// TIA Portal V17 export
// export: Created 2025-06-26T07:49:41.1534904Z, ExportSetting WithDefaults, DisplayName Totally Integrated Automation Portal, DisplayVersion V17 Update 8, DisplayName TIA Portal Openness, DisplayVersion V17 Update 8, DisplayName TIA Portal Version Control Interface, DisplayVersion V17, DisplayName STEP 7 Professional, DisplayVersion V17 Update 8, DisplayName STEP 7 Safety, DisplayVersion V17 Update 6, DisplayName WinCC Advanced, DisplayVersion V17 Update 8
FUNCTION "State2_Standby" : Void   // FC9, FBD
{ S7_Optimized_Access := 'TRUE' }
VERSION : 0.1
// stored: AutoNumber true, IsIECCheckEnabled false, SetENOAutomatically false, UDAEnableTagReadback false
   VAR_INPUT
      Active : Bool;
   END_VAR
   VAR_OUTPUT
      NextState : Bool;
      Stop : Bool;
   END_VAR
   VAR_TEMP
      NextStateConditions : Bool;
      PauseHere : Bool;
   END_VAR
   VAR_TEMP   // added for the SCL form of the ladder/FBD networks
      _w1 : Bool;
   END_VAR
BEGIN

REGION Network 1: State number
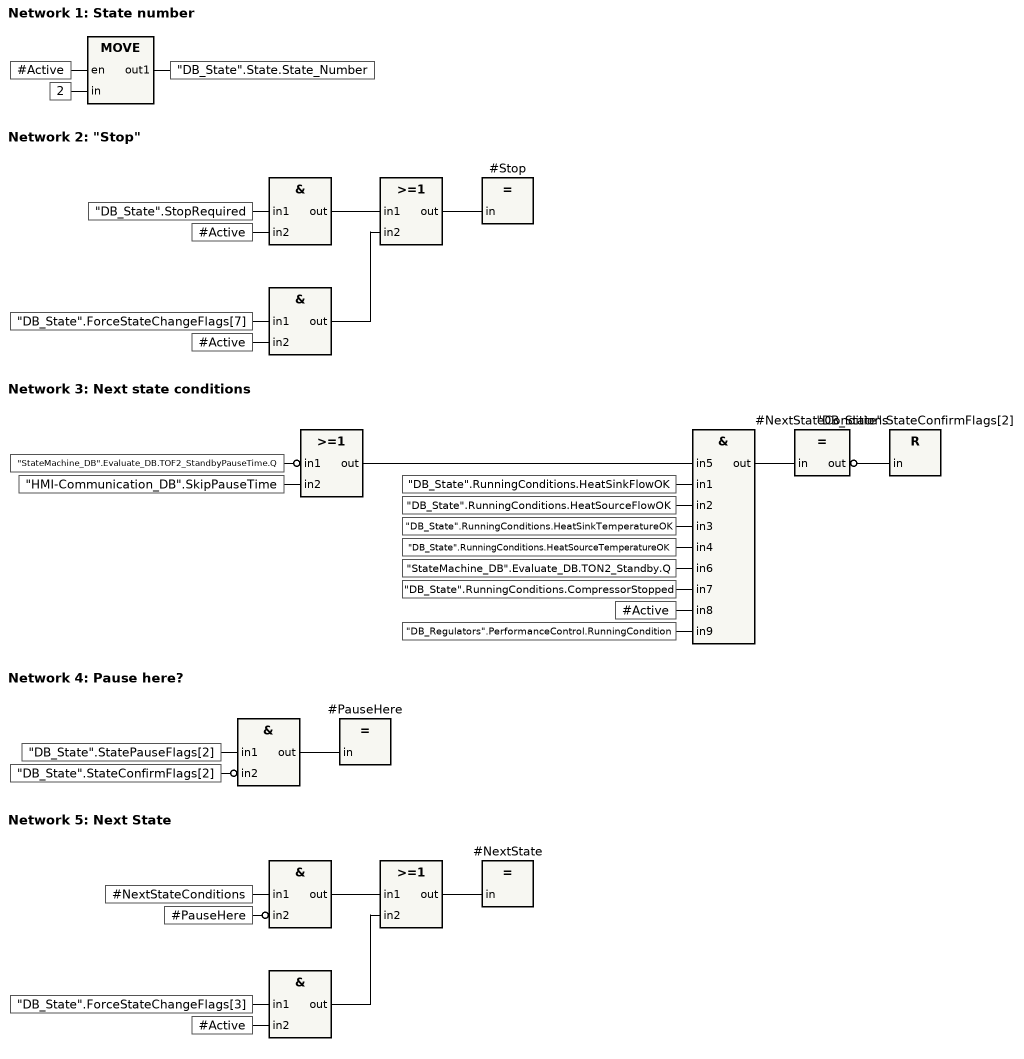
   IF #Active THEN "DB_State".State.State_Number := 2; END_IF;
END_REGION

REGION Network 2: "Stop"
   #Stop := ("DB_State".StopRequired AND #Active) OR ("DB_State".ForceStateChangeFlags[7] AND #Active);
END_REGION

REGION Network 3: Next state conditions
   #_w1 := (NOT "StateMachine_DB".Evaluate_DB.TOF2_StandbyPauseTime.Q OR "HMI-Communication_DB".SkipPauseTime) AND "DB_State".RunningConditions.HeatSinkFlowOK AND "DB_State".RunningConditions.HeatSourceFlowOK AND "DB_State".RunningConditions.HeatSinkTemperatureOK AND "DB_State".RunningConditions.HeatSourceTemperatureOK AND "StateMachine_DB".Evaluate_DB.TON2_Standby.Q AND "DB_State".RunningConditions.CompressorStopped AND #Active AND "DB_Regulators".PerformanceControl.RunningCondition;
   #NextStateConditions := #_w1;
   IF NOT #_w1 THEN "DB_State".StateConfirmFlags[2] := FALSE; END_IF;
END_REGION

REGION Network 4: Pause here?
   // Pause   Confirm  PauseHere
   // 0            0              0
   // 0            1              0
   // 1            0              1
   // 1            1              0
   #PauseHere := "DB_State".StatePauseFlags[2] AND NOT "DB_State".StateConfirmFlags[2];
END_REGION

REGION Network 5: Next State
   #NextState := (#NextStateConditions AND NOT #PauseHere) OR ("DB_State".ForceStateChangeFlags[3] AND #Active);
END_REGION
END_FUNCTION
